{attribute addProperty BoxType "EP7041-0002-0023"}
{attribute addProperty Id "ENC_Status_compactAT %I*ENC_Status_compact_DA87336C4860STM_StatusAT %I*STM_Status_64D937431620ENC_Control_compactAT %Q*ENC_Control_compact_03701F333240STM_ControlAT %Q*STM_Control_91ECC2DE1620STM_VelocityAT %Q*STM_Velocity_1D89B5C21620WcStateAT %I*WcState_F855686C1620InfoDataAT %I*InfoData_1C46E3E796120"}
{attribute addProperty CRC "192136364"}
{attribute addProperty SizeInBites "240"}
{attribute addProperty SizeInBytes "30"}
TYPE EP7041_56140984 :
STRUCT
	{attribute addProperty Name "ENC_Status_compact"}
	ENC_Status_compact : ENC_Status_compact_DA87336C;
	{attribute addProperty Name "STM_Status"}
	STM_Status : STM_Status_64D93743;
	{attribute addProperty Name "ENC_Control_compact"}
	ENC_Control_compact : ENC_Control_compact_03701F33;
	{attribute addProperty Name "STM_Control"}
	STM_Control : STM_Control_91ECC2DE;
	{attribute addProperty Name "STM_Velocity"}
	STM_Velocity : STM_Velocity_1D89B5C2;
	{attribute addProperty Name "WcState"}
	WcState : WcState_F855686C;
	{attribute addProperty Name "InfoData"}
	InfoData : InfoData_1C46E3E7;
END_STRUCT
END_TYPE

(* stored: Version 1.2.0.0, ProductVersion 3.1.4024.9
   DUT EP7041_56140984: Id {55025c6e-31b7-4ac0-a7ad-1a61275cb9da} *)
